// SIMATIC S7-200 project (STEP 7-Micro/WIN), CPU 226 REL 02.01

SYMBOL_TABLE 用户定义1
仓泵投入             I0.0
仓泵退出             I0.1
灰库高料位1           I2.7
灰库高料位2           I3.0
灰库高料位3           I3.1
进1库允许            I2.4
进2库允许            I2.5
进3库允许            I2.6
仓泵出料阀2           Q0.7
仓泵就地自动1          I1.6
气源压力上限           I1.5
仓泵压力下限           I0.6
仓泵就地料位1          I2.2
仓泵进料时间1          I1.2
仓泵出料阀1           Q0.6
仓泵输送阀1           Q0.4
仓泵排气阀1           Q0.2
仓泵进料阀1           Q0.0
仓泵就地复位1          I2.0
报警复位             I0.5
料满1              Q1.4
仓泵投入标志位          M2.4
仓泵运行标志位          M2.3
仓泵就地复位           M2.0
一号库开标志位          M8.3
二号库开标志位          M8.4
三号库开标志位          M8.5
一号库料位高报          M8.0
二号库料位高报          M8.1
三号库料位高报          M8.2
汽源压力下限           M0.7
输送阀运行超时1         M1.1
输送阀运行超时2         M1.2
堵管               M2.1
END_SYMBOL_TABLE

ORGANIZATION_BLOCK 程序块:OB1
TITLE=---------仓式输送泵程序---------
// 工业生产线上的仓泵系统，可以将物料从仓泵输送到多个库。
// [运行逻辑]
// 操作员可以通过按下仓泵投入按钮启动系统，但前提是灰库高料位传感器1、灰库高料位传感器2、灰库高料位传感器3均未检测到高料位，否则仓泵投入标志位不会置位，以防止灰库溢出。
// 系统启动后，当仓泵投入按钮被按下且仓泵运行条件满足标志为真，且至少一组灰库开标志位和进库允许信号（例如一号库开标志位和进1库允许信号）为真时，仓泵运行标志位置位，表示仓泵进入运行状态。此时，这些信号组合用于确定仓泵运行状态，但具体输送目标由外部逻辑决定。
// 进料过程开始时，仓泵运行标志位为真且进料阶段计数器值为1，系统会检查仓泵出料阀2控制是否未打开、仓泵就地自动开关1和气源压力上限传感器是否为真，只有满足这些条件，进料延时定时器1才会启动，计时30个时间单位后置位进料延时结束标志。
// 进料过程中，系统通过一系列定时器控制阀门开关：当进料延时定时器2到时、进料延时定时器3到时、进料延时定时器4到时或进料延时定时器5到时时，打开仓泵出料阀1控制；当进料延时定时器3到时或进料延时定时器11到时时，打开仓泵输送阀1控制；当进料延时定时器5到时或进料延时定时器6到时时，打开仓泵排气阀1控制；当进料延时定时器6到时时，打开仓泵进料阀1控制。
// 进料完成后，当这些定时器到时且仓泵运行标志位为真、仓泵投入标志位为假时，进料延时计数器启动，记录进料完成阶段。系统在进料开始时检查气源压力上限传感器，在特定阶段检查仓泵压力下限传感器。若输送阀运行超时标志2置位，则影响仓泵运行条件满足标志。
// 异常情况下，当进料延时定时器5到时且仓泵就地复位按钮1未按下时，报警标志置位，但只有在仓泵就地复位按钮1或报警复位按钮被按下时才会复位，恢复系统正常运行。当报警复位按钮被按下且报警标志为真时，系统准备清除异常状态。
// 操作员可以通过仓泵退出按钮复位仓泵投入标志位。此时，所有阀门如仓泵进料阀1控制、仓泵排气阀1控制、仓泵输送阀1控制、仓泵出料阀1控制、仓泵出料阀2控制保持关闭状态。仓泵就地复位按钮1用于复位仓泵就地复位标志。当仓泵就地料位传感器1检测到物料且仓泵就地复位标志为真时，系统进入复位准备状态。
// 料满指示灯1在仓泵就地料位传感器1检测到满料位且仓泵运行标志位为真且仓泵输送阀1控制未打开时点亮，提示操作员物料已满。
// 
BEGIN
Network 1 // 网络标题
// 网络注释
LD     仓泵投入:I0.0
LD     仓泵退出:I0.1
O      灰库高料位1:I2.7
O      灰库高料位2:I3.0
O      灰库高料位3:I3.1
O      SM0.1
NOT
LPS
A      仓泵投入标志位:M2.4
=      仓泵投入标志位:M2.4
LPP
ALD
O      仓泵投入标志位:M2.4
=      仓泵投入标志位:M2.4
Network 2
LDN    输送阀运行超时2:M1.2
AN     M2.6
AN     M1.7
=      M1.3
Network 3
LD     仓泵投入:I0.0
A      M1.3
LD     一号库开标志位:M8.3
A      进1库允许:I2.4
LD     二号库开标志位:M8.4
A      进2库允许:I2.5
OLD
LD     三号库开标志位:M8.5
A      进3库允许:I2.6
OLD
ALD
LDN    M1.3
O      M3.7
O      SM0.1
NOT
LPS
A      仓泵运行标志位:M2.3
=      仓泵运行标志位:M2.3
LPP
ALD
O      仓泵运行标志位:M2.3
=      仓泵运行标志位:M2.3
Network 4
LD     T47
O      M3.2
LDN    仓泵运行标志位:M2.3
ON     M1.3
O      SM0.1
O      M3.1
O      M1.6
O      M2.7
CTU    C1, 10
Network 5
LD     仓泵运行标志位:M2.3
AW=    C1, 1
LPS
AN     仓泵出料阀2:Q0.7
A      仓泵就地自动1:I1.6
A      气源压力上限:I1.5
AN     M2.5
TON    T40, 30
LPP
=      M0.6
Network 6
LDW=   C1, 2
TON    T41, 30
=      M0.1
Network 7
LDW=   C1, 3
TON    T42, 250
=      M0.2
Network 8
LDW=   C1, 4
LPS
A      仓泵压力下限:I0.6
TON    T50, 30
LPP
=      M0.0
Network 9
LDW=   C1, 5
LPS
A      仓泵投入标志位:M2.4
TON    T43, 40
LPP
=      M0.3
Network 10
LDW=   C1, 6
TON    T44, 30
=      M0.4
Network 11
LDW=   C1, 7
LPS
A      仓泵就地料位1:I2.2
TON    T45, 10
LPP
=      M0.5
Network 12
LDW=   C1, 8
TON    T46, 10
=      M1.5
Network 13
LDW=   C1, 9
=      M3.1
Network 14
LD     M3.1
O      M3.0
AN     M0.6
A      仓泵运行标志位:M2.3
=      M3.0
Network 15
LD     T45
O      仓泵进料时间1:I1.2
AW=    C1, 7
LD     T41
O      T42
O      T43
O      T44
O      T46
O      M3.6
O      M3.0
O      M3.3
O      T50
O      T40
OLD
AN     T47
TON    T47, 10
Network 16
LD     仓泵运行标志位:M2.3
AN     M2.7
EU
=      M3.2
Network 17
LD     仓泵投入标志位:M2.4
AW=    C1, 8
TON    T48, 5
AN     T48
=      M3.3
Network 18
LD     M0.1
O      M0.2
O      M0.3
O      M0.4
=      仓泵出料阀1:Q0.6
Network 19
LD     M0.2
O      M0.0
=      仓泵输送阀1:Q0.4
Network 20
LD     M0.4
O      M0.5
=      仓泵排气阀1:Q0.2
Network 21
LD     M0.5
=      仓泵进料阀1:Q0.0
Network 22
LD     M0.3
O      M0.4
O      M0.5
A      仓泵运行标志位:M2.3
AN     仓泵投入标志位:M2.4
LDN    仓泵运行标志位:M2.3
O      SM0.1
O      仓泵投入标志位:M2.4
CTU    C11, 3
Network 23
LDW=   C11, 1
LPS
TON    T49, 15
AN     T49
=      M3.6
LPP
EU
=      M1.6
Network 24
LDW=   C11, 2
EU
=      M3.7
Network 25
LD     仓泵进料时间1:I1.2
A      仓泵进料阀1:Q0.0
LD     仓泵就地料位1:I2.2
O      仓泵就地复位1:I2.0
O      报警复位:I0.5
O      SM0.1
CTU    C2, 10
Network 26
LD     M0.4
A      仓泵就地复位1:I2.0
LD     报警复位:I0.5
O      仓泵就地复位1:I2.0
O      SM0.1
NOT
LPS
A      M2.6
=      M2.6
LPP
ALD
O      M2.6
=      M2.6
Network 27
LD     C2
LD     M0.4
A      仓泵就地料位1:I2.2
OLD
EU
=      M1.4
Network 28
LD     M1.4
LD     仓泵就地复位1:I2.0
O      报警复位:I0.5
O      SM0.1
NOT
LPS
A      仓泵就地复位:M2.0
=      仓泵就地复位:M2.0
LPP
ALD
O      仓泵就地复位:M2.0
=      仓泵就地复位:M2.0
Network 29
LD     C2
A      M0.5
LD     仓泵就地料位1:I2.2
A      M0.4
OLD
LD     仓泵就地复位1:I2.0
O      报警复位:I0.5
O      SM0.1
NOT
LPS
A      M1.0
=      M1.0
LPP
ALD
O      M1.0
=      M1.0
Network 30
LD     仓泵就地料位1:I2.2
A      仓泵运行标志位:M2.3
AN     仓泵输送阀1:Q0.4
LD     M1.0
AN     SM0.5
OLD
=      料满1:Q1.4
END_ORGANIZATION_BLOCK
